# EPICS StreamDevice protocol: ioc/smApp/protocol/temp.proto
#StreamDevice protocol file for E625

ReplyTimeout = 500;
ReadTimeout = 500;
OutTerminator = CR;
InTerminator = CR;

f = 0x21;

gettemp
{
	out "#\x30\x31"; in ">%f%(\$1.VAL)f%(\$2.VAL)f%(\$3.VAL)f%(\$4.VAL)f%(\$5.VAL)f";
}

init4015
{
   out "\%\x30\x31\x30\x31\x30\x30\x30\x36\x30\x30"; in $f "%2r";
}

try
{
   out "\%\x01\x01\x00\x06\x02"; in "%1r%(\$1.VAL)1r%(\$2.VAL)1r%(\$3.VAL)1r%(\$4.VAL)1r%(\$5.VAL)1r";
}
